(*
Nazwa:			P00_Signalization
Opis:			Sygnalizacja na lini
Wersja:			v0.1
Data:			2018-10-10
Autor:			DP
Urzadzenia:		
Konfiguracja:	
Info:

*)
PROGRAM P00_Signalization
VAR

	QiLineRedSignalizationLamp 		AT %Q*:INT;				// Sygnalizacja czerwony kolor listwy LED
	QiLineGreenSignalizationLamp 	AT %Q*:INT;				// Sygnalizacja zielony kolor listwy LED	
	QiLineBlueSignalizationLamp 	AT %Q*:INT;				// Sygnalizacja niebieski kolor listwy LED		
	QiLineWhiteSignalizationLamp 	AT %Q*:INT;				// Sygnalizacja biały kolor listwy LED	
	                                            			
	QbStartLamp			 			AT %Q*:BOOL;				// Sygnalizacja startu cyklu poprzez lampkę na przyciskac
	QbResetLamp 					AT %Q*:BOOL; 				// Sygnalizacja Resetu bezpieczeństwa poprzez lampkę naprzycisku reset
	QbBuzzer						AT %Q*:BOOL;	

	QbTurnTableStartLamp			AT %Q*:BOOL;				// Sygnalizacja startu cyklu poprzez lampkę na przyciskac		
	QbTurnTableResetLamp			AT %Q*:BOOL; 				// Sygnalizacja Resetu bezpieczeństwa poprzez lampkę naprzycisku reset

	QbPucksInserterStartLamp		AT %Q*:BOOL;				// Sygnalizacja startu cyklu poprzez lampkę na przyciskac		
	QbPucksInserterResetLamp		AT %Q*:BOOL; 				// Sygnalizacja Resetu bezpieczeństwa poprzez lampkę naprzycisku reset

	
	(**BottleTransfer****)
//	QbBottleTransferRedSignalizationLamp AT %Q*:BOOL;		(*PLC.G1 robot*)		// Sygnalizacja czerwony kolor listwy LED
//	QbBottleTransferGreenSignalizationLamp AT %Q*:BOOL;		(*PLC.G1 robot*)		// Sygnalizacja zielony kolor listwy LED	
//	QbBottleTransferBlueSignalizationLamp AT %Q*:BOOL;		(*PLC.G1 robot*)		// Sygnalizacja niebieski kolor listwy LED		
//	QbBottleTransferWhiteSignalizationLamp AT %Q*:BOOL;		(*PLC.G1 robot*)		// Sygnalizacja biały kolor listwy LED	
		
	rtErrorOccure: R_TRIG;
	tofrtErrorOccure: TOF;
	TimerServiceMode: TON;
	
	
	fb1HzBlink : FB_Blink_S; // Blok wykorzystywany do wymigiwania lampki resetu
	fb5HzBlink : FB_Blink_S; // Blok wykorzystywany do wymigiwania lampki resetu
	
	
	//FB's taśma RGB
	fbRgbLedTape				: FB_RgbLedTape_EL2563;	//DMX Ul (górna taśma)
	
	//Kolor taśma LED RGB
	fbPackMlToRgb				: FB_PackMlToRgb_EL2564;//Conwersja PackML Ul w colory RGB i tryb pracy dla taśmy górnej w UL50
	
	eLastState					: E_PackMLState;
	eLastStateTemp				: E_PackMLState;
	AiProcessData				: ARRAY [1..5] OF INT;
	
	 iStep : INT := 0; // Aktualny krok efektu
    iTimer : TON; // Timer dla opóźnienia między efektami
    bTimerElapsed : BOOL := FALSE; // Flaga wskazująca, że czas minął
    iBrightness : INT := 0; // Jasność (dla efektu pulsowania)
    bIncreasing : BOOL := TRUE; // Flaga wskazująca kierunek zmiany jasności
	bTestLed: BOOL;
 	iNoteIndex : INT := 0; 
    iTimer2 : TON; 
    bTimerElapsed2 : BOOL := FALSE; 
    iDuration : TIME := T#0MS; 
    iFrequency : INT := 0; 
	
    arrM : ARRAY[1..19] OF INT := [440, 440, 440, 349, 440, 349, 440, 0, 440, 440, 440, 349, 440, 349, 440, 0, 440, 440, 440];
    arrDuration : ARRAY[1..19] OF TIME := [T#500MS, T#500MS, T#500MS, T#350MS, T#500MS, T#350MS, T#1000MS, 
                                           T#500MS, T#500MS, T#500MS, T#500MS, T#350MS, T#500MS, T#350MS, T#1000MS, 
                                           T#500MS, T#500MS, T#500MS, T#500MS];
    iMLength : INT := 19; 
	
END_VAR

(*sygnalizacja główna*)
aLamps();

ACTION aLamps:
fb1HzBlink(Tv:=T#1S);
fb5HzBlink(Tv:=T#200MS);


(*****Listwy LED*****)
(*QiLineRedSignalizationLamp:=VIS.bErrorOccure OR P00_PackML.fbPMLAuto.ePMLState = E_PMLState.ePMLState_ABORTED OR VIS.bRecipeWizardOn;
QiLineGreenSignalizationLamp:=(b2Hz AND P00_PackML.fbPMLAuto.ePMLState = E_PMLState.ePMLState_STARTING ) OR (VIS.bRecipeWizardOn AND NOT (VIS.bErrorOccure)) OR P00_PackML.fbPMLAuto.ePMLState = E_PMLState.ePMLState_STARTING OR P00_PackML.fbPMLAuto.ePMLState = E_PMLState.ePMLState_EXECUTE;
//Sterowanie Niebieskim światłem listwy led
TimerServiceMode(IN:=P00_PackML.fbPMLAuto.ePMLState = E_PMLState.ePMLState_IDLE AND P00_PackML.fbServiceMode.bOut,PT:=T#5S);
QiLineBlueSignalizationLamp:= P00_PackML.fbPMLAuto.ePMLState = E_PMLState.ePMLState_IDLE AND NOT VIS.bRecipeWizardOn AND P00_PackML.fbServiceMode.bOut;
QiLineWhiteSignalizationLamp:= (NOT QiLineRedSignalizationLamp) AND (NOT QiLineBlueSignalizationLamp) AND (NOT QiLineGreenSignalizationLamp) AND NOT VIS.bRecipeWizardOn AND NOT (P00_PackML.fbPMLAuto.ePMLState = E_PMLState.ePMLState_EXECUTE); 
*)
//Vasyl 03.10 Reset nie mruga póki nie skończy się timer tonbFirstCycle.Q w ACT_SafetyFirstResetDelay
(*****Przyciski*****)
QbStartLamp := (((	P00_PackML.fbPMLAuto.ePMLState = Tc3_PackML.E_PMLState.ePMLState_IDLE  OR P00_PackML.fbPMLAuto.ePMLState = Tc3_PackML.E_PMLState.ePMLState_SUSPENDED) AND 
               		P00_PackML.fbPMLModeManager.eModeStatus = Tc3_PackML.E_PMLUnitMode.ePMLUnitMode_AUTOMATIC AND (P00_PackML.bStationsAreReady AND NOT P00_PackML.bAtLeastOneOfTheStationsNeedHoming)) AND fb1HzBlink.Q);
			   
QbResetLamp:=NOT IbEmergencyStop AND b1Hz AND P00_PackML.tonbFirstCycle.Q;

QbTurnTableStartLamp	:=	QbStartLamp;
QbTurnTableResetLamp	:=	QbResetLamp;

QbPucksInserterStartLamp:=	QbStartLamp;
QbPucksInserterResetLamp:=	QbResetLamp;

(*****Buzzer********)
rtErrorOccure 			(CLK :=VIS.bErrorOccure, Q=>);
tofrtErrorOccure 		(IN := rtErrorOccure.Q , PT := T#5S);
IF NOT bTestLed THEN
QbBuzzer 			:=	(P00_PackML.fbPMLAuto.ePMLState = Tc3_PackML.E_PMLState.ePMLState_STARTING AND b1Hz AND NOT P00_PackML.tonStarting.Q) OR bSoftAlarm OR (tofrtErrorOccure.Q AND b1Hz);
END_IF

(*Warningi*)
IF (P08_CapFeeder.fbCapFeeder.bWarning1 OR P01_BottleFeeder.fbBottleFeeder.bWarning1) AND P00_PackML.fbPMLAuto.ePMLState = Tc3_PackML.E_PMLState.ePMLState_EXECUTE THEN
	(*QiLineRedSignalizationLamp			:= TRUE;
	QiLineGreenSignalizationLamp			:= FALSE;
	QiLineBlueSignalizationLamp				:= TRUE;
	QiLineWhiteSignalizationLamp			:= FALSE;*)
END_IF


IF VIS.bWeighingForm AND b1Hz AND P00_PackML.fbPMLAuto.ePMLState = Tc3_PackML.E_PMLState.ePMLState_EXECUTE THEN
	(*QiLineRedSignalizationLamp				:= FALSE; 
	QiLineGreenSignalizationLamp			:= TRUE;
	QiLineBlueSignalizationLamp				:= TRUE;
	QiLineWhiteSignalizationLamp			:= FALSE;*)
END_IF


fbPackMlToRgb(
					ePackMLState		:= P00_PackML.fbPMLAuto.ePMLState,
					ePackMLMode			:= P00_PackML.fbPMLModeManager.eModeStatus, 
					eLastState			:= eLastState, 
					nDelayButtonBlinkIn	:= , 
					bStopViaOut			:= , 
					bWarning			:= VIS.uliWarningOccure>0, 
					bHoming				:= Gvl.bHoming, 
					bWeighingForm		:= VIS.bWeighingForm,
					bLowMaterialInExecute:=	P00_Visualization.tonNoFormsBeforeDispencers.Q OR 
											P00_PackML.tonCycleBadBottleConveyorFullSensor.Q OR P16_LabelMachine.tonLabelMachineFullSensorInfo.Q OR
											P06_LidFeeder.bLidFeederWarning1 OR P06_LidFeeder.bLidFeederWarning2 OR
											P06_WickFeeder.fbWickFeederSt.bWarning,
					nCh1Red				=> ,
					nCh2Green			=> ,
					nCh3Blue			=> , 
					nCh4White			=> , 
					nCh5Reserve=> , 
					bBlink=> , 
					bBlink2Colors=> , 					
					bHorn=> , 
					bStartButtonLampOut=> );

fbRgbLedTape(	 
				   	bEnable				:= TRUE,
					nCh1Red				:= fbPackMlToRgb.nCh1Red,
					nCh2Green			:= fbPackMlToRgb.nCh2Green,
					nCh3Blue			:= fbPackMlToRgb.nCh3Blue,
					nCh4White			:= fbPackMlToRgb.nCh4White,
					nCh5Reserve			:= fbPackMlToRgb.nCh5Reserve,
					bBlink				:= fbPackMlToRgb.bBlink,
					bBlink2Colors		:= fbPackMlToRgb.bBlink2Colors,					
					nDelayBlink 		:= 1,
					nMaxBlinkValue		:= 32766,
					AiProcessData		:= AiProcessData);
IF NOT bTestLed THEN		
	QiLineRedSignalizationLamp 				:= AiProcessData[1];  
	QiLineGreenSignalizationLamp 			:= AiProcessData[2];
	QiLineBlueSignalizationLamp 			:= AiProcessData[3];
	QiLineWhiteSignalizationLamp 			:= AiProcessData[4];
ELSE
		// Logika sterowania
	iTimer(IN := TRUE, PT := T#500MS); // Timer ustawiony na 500 ms
	bTimerElapsed := iTimer.Q;
	
	IF bTimerElapsed THEN
		iTimer(IN := FALSE); // Resetowanie timera
		iTimer(IN := TRUE);  // Restart timera
		
		CASE iStep OF
			0: // Czerwony
				QiLineRedSignalizationLamp := 10000; // Maksymalna jasność
				QiLineGreenSignalizationLamp := 0;
				QiLineBlueSignalizationLamp := 0;
				QiLineWhiteSignalizationLamp := 0;
			1: // Zielony
				QiLineRedSignalizationLamp := 0;
				QiLineGreenSignalizationLamp := 10000; // Maksymalna jasność
				QiLineBlueSignalizationLamp := 0;
				QiLineWhiteSignalizationLamp := 0;
			2: // Niebieski
				QiLineRedSignalizationLamp := 0;
				QiLineGreenSignalizationLamp := 0;
				QiLineBlueSignalizationLamp := 10000; // Maksymalna jasność
				QiLineWhiteSignalizationLamp := 0;
			3: // Biały
				QiLineRedSignalizationLamp := 0;
				QiLineGreenSignalizationLamp := 0;
				QiLineBlueSignalizationLamp := 0;
				QiLineWhiteSignalizationLamp := 10000; // Maksymalna jasność
			4: // Pulsowanie jasności
				IF bIncreasing THEN
					iBrightness := iBrightness + 1000;
					IF iBrightness >= 10000 THEN
						bIncreasing := FALSE;
					END_IF
				ELSE
					iBrightness := iBrightness - 1000;
					IF iBrightness <= 0 THEN
						bIncreasing := TRUE;
					END_IF
				END_IF
				QiLineRedSignalizationLamp := iBrightness;
				QiLineGreenSignalizationLamp := iBrightness;
				QiLineBlueSignalizationLamp := iBrightness;
				QiLineWhiteSignalizationLamp := iBrightness;
		END_CASE;
		
		iStep := iStep + 1;
		IF iStep > 4 THEN
			iStep := 0; // Powrót do pierwszego kroku
		END_IF;
	END_IF;
	
    // Timer nuty
    iTimer2(IN := TRUE, PT := iDuration); 
    bTimerElapsed2 := iTimer2.Q;

    IF bTimerElapsed2 THEN

        iTimer2(IN := FALSE); // Reset timera
        iTimer2(IN := TRUE);  // Restart timera
        iNoteIndex := iNoteIndex + 1;
       
        IF iNoteIndex > iMLength THEN
            iNoteIndex := 1;
        END_IF;

        // Ustawienie częstotliwości i czasu trwania 
        iFrequency := arrM[iNoteIndex];
        iDuration := arrDuration[iNoteIndex];

        // Generowanie dźwięku na buzzerze
        IF iFrequency > 0 THEN
            QbBuzzer := TRUE; // Aktywacja buzzera
        ELSE
            QbBuzzer := FALSE; // Pauza
        END_IF;
    END_IF;	
		
END_IF

(*
fbRgbLedTape(	 
				   	bEnable				:= TRUE,
					nCh1Red				:= 0,
					nCh2Green			:= 32000,
					nCh3Blue			:= 10000,
					nCh4White			:= 0,
					nCh5Reserve			:= 0,
					bBlink				:= FALSE,
					bBlink2Colors		:= TRUE,					
					nDelayBlink 		:= 1,
					nMaxBlinkValue		:= 32766,
					AiProcessData		:= AiProcessData);
			
QiLineRedSignalizationLamp 				:= 	AiProcessData[1];
QiLineGreenSignalizationLamp 			:= 	AiProcessData[2];
QiLineBlueSignalizationLamp 			:= 	AiProcessData[3];
QiLineWhiteSignalizationLamp 			:= 	AiProcessData[4];
*)
END_ACTION

END_PROGRAM

(* stored: Version 1.1.0.1, ProductVersion 3.1.4026.13, FileIdentifier b2cbb4b26c6a25309f4412dee5e63901f5372872, FileSignature 3baf967b37d10bfb20b2687e11c331d9496b6321321c560b6c50115cff8748e4b6acfc3659e07ceb55e4d8ad45697ee362878e080734cc8dd2e68df5eff9ac38d1e21565d50ac2454aba9cb6f909384d21c6842f85d7ba405f0fc819881eb0b528619551ebd8a148fba31328db6482c187685f445067739929dadee5d569485ff255061a8476792c9d7ae985c2a340e0fc0ae35e7af44319df8f052a970450fb1685beda69810645ad8760801ea52302904585f058761c1430a9c9cb98df254cb3d77196ebffaff399a523fa6934c66ef1faed6e6ca0db9c7bd30c64a1332a3c12c05f5b16281cfb6d8d3d0cb1af091f6823d1402c7516eb19bbd93c761b3ed0
   POU P00_Signalization: Id {3eec4104-0b2f-458a-864a-1eb1ed28a562}, SpecialFunc None
   Action aLamps: Id {226ec791-019e-4967-a707-6de482b85d3d} *)
